FUNCTION_BLOCK MetalSaltDosingActuators (* CAT Function Block Type *)
  (* Standard: 61499-2 *)
  (* Version 0.0, 7/9/2026, Schneider Electric, template *)
  PACKAGE SE.Nereda;
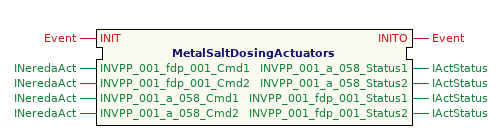
  EVENT_INPUT
    INIT;
  END_EVENT
  EVENT_OUTPUT
    INITO;
  END_EVENT
  SOCKETS
    INVPP_001_fdp_001_Cmd1 : INeredaAct;
    INVPP_001_fdp_001_Cmd2 : INeredaAct;
    INVPP_001_a_058_Cmd1 : INeredaAct;
    INVPP_001_a_058_Cmd2 : INeredaAct;
  END_SOCKETS
  PLUGS
    INVPP_001_a_058_Status1 : IActStatus;
    INVPP_001_a_058_Status2 : IActStatus;
    INVPP_001_fdp_001_Status1 : IActStatus;
    INVPP_001_fdp_001_Status2 : IActStatus;
  END_PLUGS
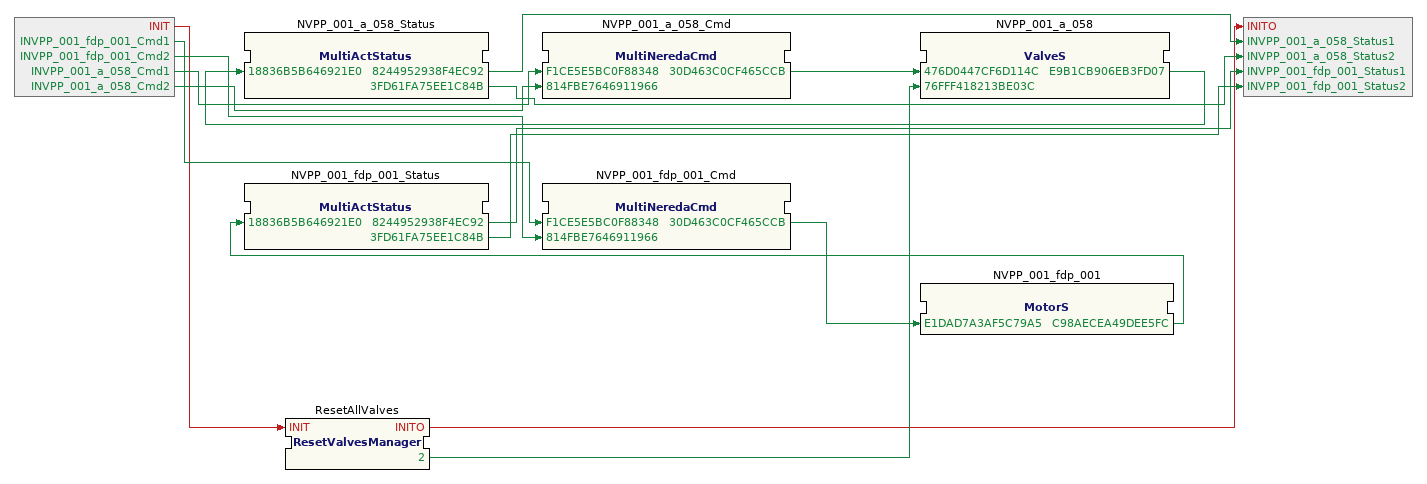
  (* 01 - FUNCTIONNAL INPUT INTERFACE *)
  (* 00 - INITIALIZATION *)
  (* 05 - LOGIC *)
  (* 06 - HMI INTERFACE *)
  (* 03 - FIELD INTERFACE *)
  (* 02 - FUNCTIONNAL OUTPUT INTERFACE *)
  (* Actuators Status *)
  (* 04 - CHILDREN *)
  (* 4A - TYPICALS *)
  (* Actuators Command *)
  (* Reset All Actuators *)
  FBS
    ResetAllValves : ResetValvesManager;
    NVPP_001_a_058 : ValveS;
    NVPP_001_a_058_Status : MultiActStatus;
    NVPP_001_fdp_001_Status : MultiActStatus;
    NVPP_001_a_058_Cmd : MultiNeredaCmd;
    NVPP_001_fdp_001_Cmd : MultiNeredaCmd;
    NVPP_001_fdp_001 : MotorS;
  END_FBS
  EVENT_CONNECTIONS
    INIT TO ResetAllValves.INIT;
    ResetAllValves.INITO TO INITO;
  END_CONNECTIONS
  ADAPTER_CONNECTIONS
    NVPP_001_a_058_Cmd.30D463C0CF465CCB TO NVPP_001_a_058.476D0447CF6D114C;
    NVPP_001_fdp_001_Cmd.30D463C0CF465CCB TO NVPP_001_fdp_001.E1DAD7A3AF5C79A5;
    NVPP_001_a_058.E9B1CB906EB3FD07 TO NVPP_001_a_058_Status.18836B5B646921E0;
    NVPP_001_fdp_001.C98AECEA49DEE5FC TO NVPP_001_fdp_001_Status.18836B5B646921E0;
    INVPP_001_a_058_Cmd1 TO NVPP_001_a_058_Cmd.F1CE5E5BC0F88348;
    INVPP_001_a_058_Cmd2 TO NVPP_001_a_058_Cmd.814FBE7646911966;
    INVPP_001_fdp_001_Cmd1 TO NVPP_001_fdp_001_Cmd.F1CE5E5BC0F88348;
    INVPP_001_fdp_001_Cmd2 TO NVPP_001_fdp_001_Cmd.814FBE7646911966;
    NVPP_001_a_058_Status.8244952938F4EC92 TO INVPP_001_a_058_Status1;
    NVPP_001_a_058_Status.3FD61FA75EE1C84B TO INVPP_001_a_058_Status2;
    NVPP_001_fdp_001_Status.8244952938F4EC92 TO INVPP_001_fdp_001_Status1;
    NVPP_001_fdp_001_Status.3FD61FA75EE1C84B TO INVPP_001_fdp_001_Status2;
    ResetAllValves.2 TO NVPP_001_a_058.76FFF418213BE03C;
  END_CONNECTIONS
END_FUNCTION_BLOCK
